// TIA Portal V19 export
DATA_BLOCK "dataBlockGlobal"   // DB555
{ S7_Optimized_Access := 'TRUE' }
// stored: AutoNumber false, MemoryReserve 100
   VAR
      new : Array[0..99] of Byte;
   END_VAR
BEGIN
END_DATA_BLOCK
